{attribute addProperty BoxType "EL4028-0000-0018"}
{attribute addProperty Id "AO_Output_ChannelAT %Q*ARRAY[0..7] OF AO_Output_Channel_F57FA4F9128160WcStateAT %I*WcState_64F6A8C6810InfoDataAT %I*InfoData_BC63D37F80100"}
{attribute addProperty CRC "683782063"}
{attribute addProperty SizeInBites "216"}
{attribute addProperty SizeInBytes "27"}
TYPE EL4028_02F9C07C :
STRUCT
	{attribute addProperty Name "AO_Output_Channel"}
	AO_Output_Channel : ARRAY[0..7] OF AO_Output_Channel_F57FA4F9;
	{attribute addProperty Name "WcState"}
	WcState : WcState_64F6A8C6;
	{attribute addProperty Name "InfoData"}
	InfoData : InfoData_BC63D37F;
END_STRUCT
END_TYPE

(* stored: Version 1.2.0.0, ProductVersion 3.1.4024.9
   DUT EL4028_02F9C07C: Id {548ab7fc-8a7d-44f5-9bff-fd0a7f1f562f} *)
